{attribute addProperty BoxType "EK1100-0000-0018"}
{attribute addProperty Id "Beckhoff_ELM3xxxEK1122Beckhoff_ELM3xxxEK1122_52A3E13B162A_0001_ELM3002_0000_0016ELM3002_1C598C2535244A_0002_ELM3002_0000_0017ELM3002_1C598C2535244A_0003_ELM3002_0000_0018ELM3002_1C598C2535244A_0004_ELM3004_0000_0016ELM3004_EF18820948060A_0005_ELM3004_0000_0017ELM3004_EF18820948060A_0006_ELM3004_0000_0018ELM3004_EF18820948060A_0007_ELM3004_0000_0019ELM3004_EF18820948060"}
{attribute addProperty CRC "1147131006"}
{attribute addProperty SizeInBites "2992"}
{attribute addProperty SizeInBytes "374"}
TYPE Beckhoff_ELM3xxx_445FD47E EXTENDS EK1100_179A0949 :
STRUCT
	{attribute addProperty Name "Beckhoff_ELM3xxxEK1122"}
	Beckhoff_ELM3xxxEK1122 : Beckhoff_ELM3xxxEK1122_52A3E13B;
	{attribute addProperty Name "A_0001_ELM3002_0000_0016"}
	A_0001_ELM3002_0000_0016 : ELM3002_1C598C25;
	{attribute addProperty Name "A_0002_ELM3002_0000_0017"}
	A_0002_ELM3002_0000_0017 : ELM3002_1C598C25;
	{attribute addProperty Name "A_0003_ELM3002_0000_0018"}
	A_0003_ELM3002_0000_0018 : ELM3002_1C598C25;
	{attribute addProperty Name "A_0004_ELM3004_0000_0016"}
	A_0004_ELM3004_0000_0016 : ELM3004_EF188209;
	{attribute addProperty Name "A_0005_ELM3004_0000_0017"}
	A_0005_ELM3004_0000_0017 : ELM3004_EF188209;
	{attribute addProperty Name "A_0006_ELM3004_0000_0018"}
	A_0006_ELM3004_0000_0018 : ELM3004_EF188209;
	{attribute addProperty Name "A_0007_ELM3004_0000_0019"}
	A_0007_ELM3004_0000_0019 : ELM3004_EF188209;
END_STRUCT
END_TYPE

(* stored: Version 1.2.0.0, ProductVersion 3.1.4024.9
   DUT Beckhoff_ELM3xxx_445FD47E: Id {986b7917-d164-42b2-ba36-776122c79cc0} *)
